(* Logix 5000 project; controller FRIST_EXAMPLE Emulate 5570 rev 19.11; software revision 19.01 *)

TASK MainTask (continuous, watchdog 500 ms) : MainProgram

MODULES
   Local : Emulate 5570 (ICP 2, rev 19.11)
       : 1756-IB32 (ICP 3, rev 3.1, Input RPI 20 ms)   // DG-INPUT
       : vendor 1 type 7 code 8 (ICP 4, rev 3.1, Output RPI 20 ms)
       : 1756-IF6I (ICP 5, rev 1.1, Input RPI 100 ms)
       : 1756-OF8 (ICP 6, rev 1.1, Output RPI 12 ms)
END_MODULES

VAR_GLOBAL   (* controller tags *)
   CMD_MT01 : BOOL;
   DESLIGA : BOOL := 1;
   LIGA : BOOL;
END_VAR

PROGRAM MainProgram   (* main routine MainRoutine *)
VAR
   BT_DESLIGA : BOOL;
   BT_LIGA : BOOL;
   MOTOR : BOOL[32];
   T_PARADA : TIMER;
   T_PARTIDA : TIMER := (PRE := 10000);
END_VAR

ROUTINE MainRoutine   (* ladder *)
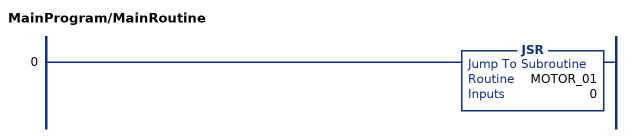
   0: JSR(MOTOR_01,0);
END_ROUTINE

ROUTINE MOTOR_01   (* ladder *)
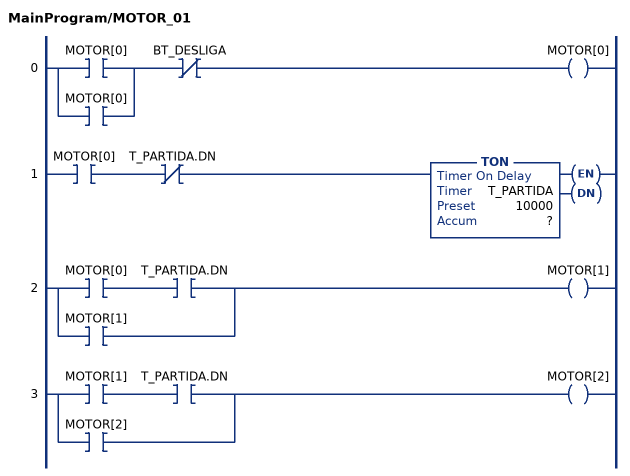
   0: [XIC(MOTOR[0]) ,XIC(MOTOR[0]) ]XIO(BT_DESLIGA)OTE(MOTOR[0]);
   1: XIC(MOTOR[0])XIO(T_PARTIDA.DN)TON(T_PARTIDA,?,?);
   2: [XIC(MOTOR[0]) XIC(T_PARTIDA.DN) ,XIC(MOTOR[1]) ]OTE(MOTOR[1]);
   3: [XIC(MOTOR[1]) XIC(T_PARTIDA.DN) ,XIC(MOTOR[2]) ]OTE(MOTOR[2]);
END_ROUTINE
END_PROGRAM
